// SIMATIC S7-200 project (STEP 7-Micro/WIN), CPU 224 REL 01.10

ORGANIZATION_BLOCK MAIN:OB1
TITLE=我做了一个PLC程序包含啤酒发酵控制模。涉及的设备包括温度传感器、压力传感器和电磁阀。 系统通过温度传感器和压力传感器实时监测发酵罐的状态，将数据存储到暂存区，并转换为实数数据用于计算。系统通过预设的传感器数据处理流程，确保传感器读数适用于后续计算。系统支持多个发酵罐运行，以发酵罐1为例，发酵罐状态表示其运行状态，值在0到4之间，0表示停止，1到4分别对应不同的发酵阶段，如主教阶段。通过条件判断，系统只识别这些运行状态并据此操作。在每个阶段，系统根据工艺需求计算温度设定值，用于满足发酵工艺的温度条件。温度控制通过PID算法实现，依赖比例系数、积分时间和微分时间计算控制输出。这些参数根据发酵罐特性预设，以支持稳定的温度控制。计算结果驱动电磁阀开关，调节发酵罐的温度。为实现精确控制，系统使用电磁阀开关定时器和电磁阀关闭定时器，分别以开启预设时间和关闭预设时间为基准，控制开关时间。
BEGIN
Network 1 // 网络标题
// 网络注释
LD     SM0.0
LPS
MOVW   AIW0, VW10
AENO
MOVW   AIW2, VW12
AENO
MOVW   AIW4, VW14
LRD
MOVW   AIW6, VW16
AENO
MOVW   AIW8, VW18
LRD
MOVW   AIW10, VW20
AENO
MOVW   AIW12, VW22
AENO
MOVW   AIW14, VW24
LRD
MOVW   AIW16, VW26
AENO
MOVW   AIW18, VW28
LRD
MOVW   AIW20, VW30
AENO
MOVW   AIW22, VW32
AENO
MOVW   AIW24, VW34
LPP
MOVW   AIW26, VW36
AENO
MOVW   AIW28, VW38
Network 2
LD     SM0.0
LPS
ITD    VW10, VD40
AENO
ITD    VW12, VD44
AENO
ITD    VW14, VD48
AENO
ITD    VW16, VD52
LRD
ITD    VW18, VD56
AENO
ITD    VW20, VD60
AENO
ITD    VW22, VD64
AENO
ITD    VW24, VD68
LPP
ITD    VW26, VD72
AENO
ITD    VW28, VD76
Network 3
// 整数转换成实数(一个发酵罐为例)
LD     SM0.0
LPS
DTR    VD40, VD100
AENO
DTR    VD44, VD104
AENO
DTR    VD48, VD108
LRD
DTR    VD52, VD112
AENO
DTR    VD56, VD116
LRD
DTR    VD60, VD120
AENO
DTR    VD64, VD124
AENO
DTR    VD68, VD128
LPP
DTR    VD72, VD132
AENO
DTR    VD76, VD136
Network 4
// vb1000 发酵罐1状态 vb1002 发酵罐2状态 0状态，停止温控，不计时
LD     SM0.0
LDB=   VB1000, 0
OB=    VB1002, 0
OB=    VB1004, 0
ALD
JMP    1
Network 5
// 主教阶段
LD     SM0.0
LPS
AB=    VB1000, 1
S      M10.0, 1
R      M10.1, 1
R      M10.2, 1
R      M10.3, 1
LPP
AB=    VB1002, 1
S      M11.0, 1
R      M11.1, 1
R      M11.2, 1
R      M11.3, 1
Network 6
LD     SM0.0
LPS
AB=    VB1000, 2
S      M10.1, 1
R      M10.0, 1
R      M10.2, 1
R      M10.3, 1
LPP
AB=    VB1002, 2
S      M11.1, 1
R      M11.0, 1
R      M11.2, 1
R      M11.3, 1
Network 7
// //其余的都在这个基础上改把
// 
LD     SM0.0
LPS
AB=    VB1000, 3
S      M10.2, 1
R      M10.0, 1
R      M10.1, 1
R      M10.3, 1
LPP
AB=    VB1002, 3
S      M11.2, 1
R      M11.0, 1
R      M11.1, 1
R      M11.3, 1
Network 8
LD     SM0.0
LPS
AB=    VB1000, 4
S      M10.3, 1
R      M10.0, 1
R      M10.1, 1
R      M10.2, 1
LPP
AB=    VB1002, 4
S      M11.3, 1
R      M11.0, 1
R      M11.1, 1
R      M11.2, 1
Network 9
LD     SM0.0
LPS
A      M10.0
MOVB   1, VB2000
AENO
CALL   计时:SBR0
LRD
A      M10.1
MOVB   2, VB2000
AENO
CALL   计时:SBR0
LPP
A      M10.2
MOVB   3, VB2000
AENO
CALL   计时:SBR0
Network 10
LBL    1
Network 11
// 计算温度设定值，由此引出 M10.1 ,M10.2 ,M10.3 这几个阶段，都是如此
// 
// 另外 在加一只发酵罐
LD     SM0.0
A      M10.0
LPS
MOVR   VD200, VD1200
AENO
MOVR   VD204, VD1204
AENO
=      L63.7
LPP
MOVR   VD208, VD1208
AENO
MOVR   VD212, VD1212
AENO
O      L63.7
MOVW   VW300, VW1216
AENO
CALL   设定值:SBR1
Network 12
// PID控制  kp                                                              ti                                                       td
LD     SM0.0
MOVR   VD220, VD1220
AENO
MOVR   VD224, VD1224
AENO
MOVR   VD228, VD1228
AENO
MOVR   VD232, VD1232
Network 13
//     en  ----> en-1                                                                               M ----->M-1
LD     SM0.0
MOVR   VD1236, VD1240
AENO
MOVR   VD1272, VD1276
Network 14
LD     SM0.4
EU
CALL   PID计算:SBR2
Network 15
// kongzhi diancifa 
MOVR   VD1272, VD1300
AENO
MOVR   VD1300, VD1312
AENO
*R     VD1304, VD1312
AENO
MOVD   VD1312, VD1320
AENO
-D     VD1304, VD1320
AENO
*R     600.0, VD1312
AENO
AN     T37
=      Q0.1
Network 16
LD     Q0.1
LPS
EU
MOVD   VD1312, VD1316
LPP
ED
MOVD   VD1320, VD1324
*D     +600, VD1324
Network 17
LD     Q0.1
TON    T37, VW1318
Network 18
LDN    Q0.1
TON    T38, VW1324
R      T37, 1
END_ORGANIZATION_BLOCK

SUBROUTINE_BLOCK 计时:SBR0
TITLE=子例行程序注释
BEGIN
Network 1 // 网络标题
// 网络注释
LD     SM0.0
CALL   计时:SBR0
END_SUBROUTINE_BLOCK

SUBROUTINE_BLOCK 设定值:SBR1
TITLE=子例行程序注释
BEGIN
Network 1 // 网络标题
// 网络注释温度                                                   时间                                                                 除数 谢率
LD     SM0.0
MOVR   VD1204, VD1220
AENO
-R     VD1200, VD1220
AENO
MOVR   VD1212, VD1224
AENO
-R     VD1208, VD1224
AENO
MOVR   VD1220, VD1228
/R     VD1224, VD1228
Network 2
//                                                                                                   设定温度
LD     SM0.0
MOVR   VD1228, VD1232
AENO
*R     VD1216, VD1232
AENO
MOVR   VD1232, VD1236
+R     VD1200, VD1236
END_SUBROUTINE_BLOCK

SUBROUTINE_BLOCK PID计算:SBR2
TITLE=子例行程序注释
BEGIN
Network 1 // 网络标题
// 网络注释     正反作用标志M20.0      1正0反 
LD     SM0.0
LPS
A      M20.0
MOVR   VD1244, VD1236
-R     VD1248, VD1236
LPP
AN     M20.0
MOVR   VD1248, VD1236
-R     VD1244, VD1236
Network 2
// en--en-1                                                      kp(en - en-1)
LD     SM0.0
MOVR   VD1236, VD1252
AENO
-R     VD1240, VD1252
AENO
*R     VD1220, VD1252
Network 3
// ts* en                                                                                ts* en/ti                                                        ts * en * kp/ti
LD     SM0.0
MOVR   VD1232, VD1256
AENO
*R     VD1236, VD1256
AENO
/R     VD1224, VD1256
AENO
*R     VD1220, VD1256
Network 4
// vn+ vn-2                                                                      Vn + Vn-2   --2* Vn-1
LD     SM0.0
MOVR   VD1248, VD1260
AENO
+R     VD1268, VD1260
AENO
-R     VD1264, VD1260
AENO
-R     VD1264, VD1260
Network 5
//    (Vn + Vn-2   --2* Vn-1)  * KP                       (Vn + Vn-2   --2* Vn-1)  * KP * TS            (Vn + Vn-2   --2* Vn-1)  * KP * TS/Td
LD     SM0.0
*R     VD1220, VD1260
AENO
*R     VD1232, VD1260
AENO
/R     VD1228, VD1260
Network 6
LD     SM0.0
MOVR   0.0, VD1272
AENO
+R     VD1260, VD1272
AENO
+R     VD1256, VD1272
AENO
+R     VD1252, VD1272
AENO
+R     VD1276, VD1272
Network 7
//        pv1---->pv2                                                   pv---pv1
LD     SM0.0
MOVR   VD1264, VD1268
AENO
MOVR   VD1248, VD1264
END_SUBROUTINE_BLOCK
